// TIA Portal V17 export
// export: Created 2024-08-26T21:10:51.5472391Z, ExportSetting WithDefaults, DisplayName Totally Integrated Automation Portal, DisplayVersion V17 Update 7, DisplayName TIA Portal Openness, DisplayVersion V17 Update 7, DisplayName TIA Portal Version Control Interface, DisplayVersion V17, DisplayName SINAMICS Startdrive Advanced, DisplayVersion V17 SP2, DisplayName SINAMICS Startdrive G110M, G120, G120C, G120D, G120P, G115D, DisplayVersion V17 SP2, DisplayName SINAMICS Startdrive G130, G150, S120, S150, SINAMICS MV, S210, DisplayVersion V17 SP2, DisplayName STEP 7 Professional, DisplayVersion V17 Update 7, DisplayName STEP 7 Safety, DisplayVersion V17 Update 6, DisplayName WinCC Advanced / Unified PC, DisplayVersion V17 Update 7
FUNCTION "MODE" : Void   // FC4, LAD
{ S7_Optimized_Access := 'TRUE' }
VERSION : 0.1
// stored: AutoNumber true, IsIECCheckEnabled false, SetENOAutomatically false, UDAEnableTagReadback false
   VAR_TEMP
      f7 : Bool;
      BF7 : Bool;
   END_VAR
BEGIN

REGION Network 1: MODE CHANGE
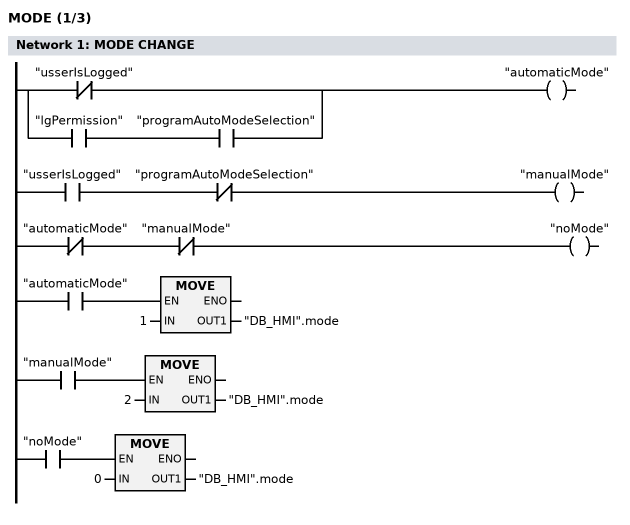
   RUNG wire#powerrail
      I_Contact( "usserIsLogged" )
      wire#w1
      Coil( "automaticMode" )
   END_RUNG
   RUNG wire#powerrail
      Contact( "lgPermission" )
      Contact( "programAutoModeSelection" )
   END_RUNG wire#w1
   RUNG wire#powerrail
      Contact( "usserIsLogged" )
      I_Contact( "programAutoModeSelection" )
      Coil( "manualMode" )
   END_RUNG
   RUNG wire#powerrail
      I_Contact( "automaticMode" )
      I_Contact( "manualMode" )
      Coil( "noMode" )
   END_RUNG
   RUNG wire#powerrail
      Contact( "automaticMode" )
      Move(in := 1, out1 => "DB_HMI".mode)
   END_RUNG
   RUNG wire#powerrail
      Contact( "manualMode" )
      Move(in := 2, out1 => "DB_HMI".mode)
   END_RUNG
   RUNG wire#powerrail
      Contact( "noMode" )
      Move(in := 0, out1 => "DB_HMI".mode)
   END_RUNG
   // the same network as SCL:
   "automaticMode" := NOT "usserIsLogged" OR ("lgPermission" AND "programAutoModeSelection");
   "manualMode" := "usserIsLogged" AND NOT "programAutoModeSelection";
   "noMode" := NOT "automaticMode" AND NOT "manualMode";
   IF "automaticMode" THEN "DB_HMI".mode := 1; END_IF;
   IF "manualMode" THEN "DB_HMI".mode := 2; END_IF;
   IF "noMode" THEN "DB_HMI".mode := 0; END_IF;
END_REGION

REGION Network 2: MODEL SELECTION
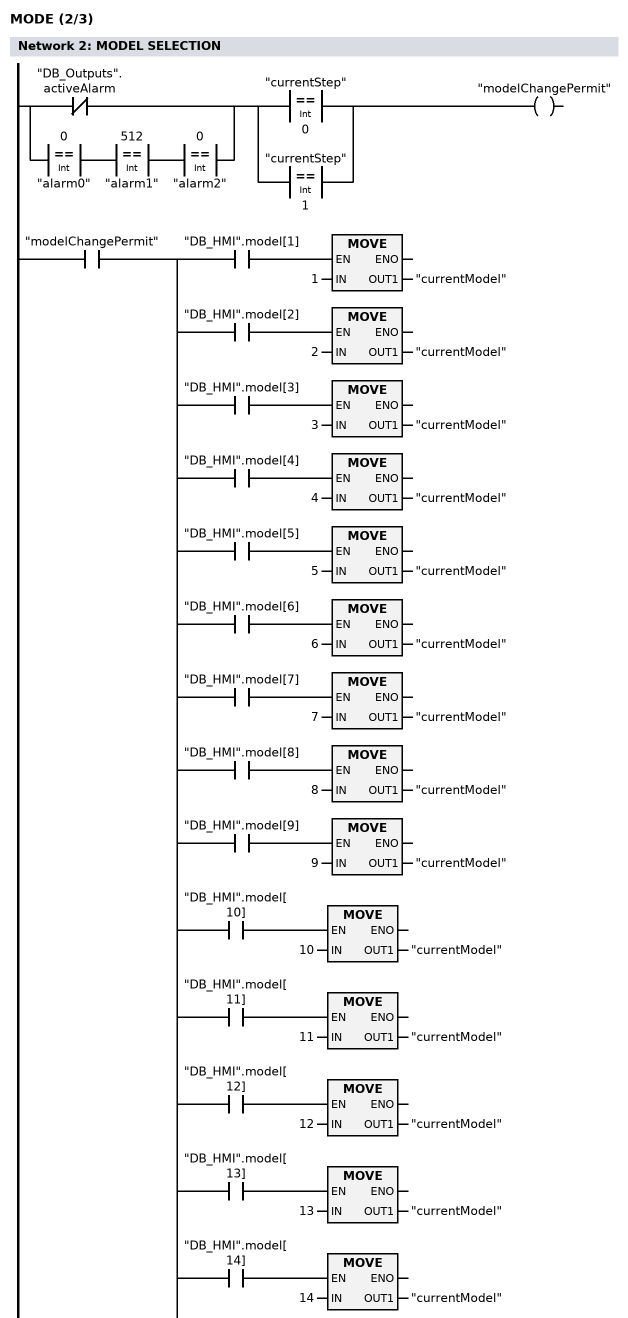
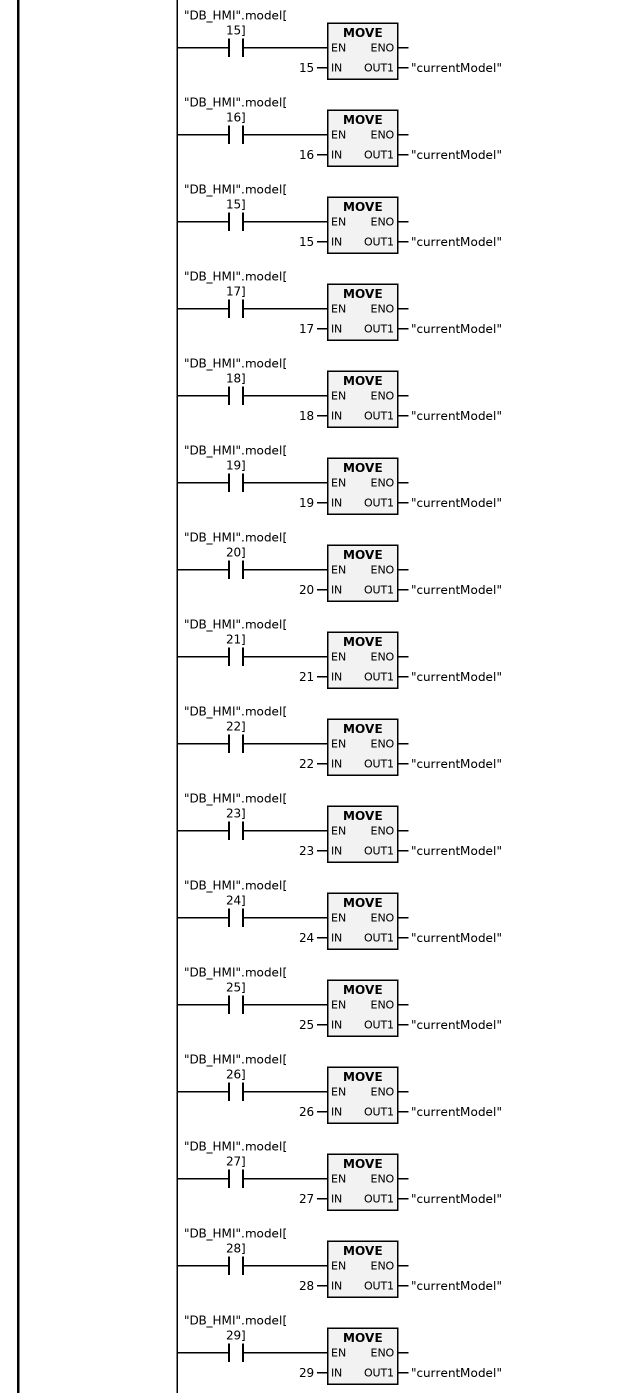
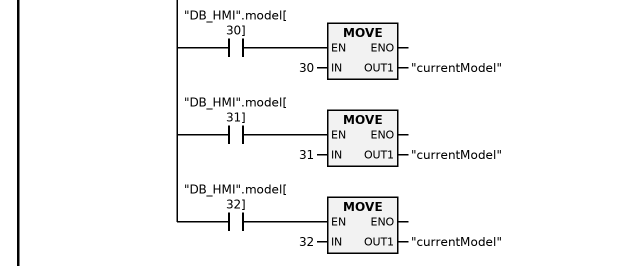
   RUNG wire#powerrail
      I_Contact( "DB_Outputs".activeAlarm )
      wire#w1
      { S7_Templates := "SrcType := Int" } EQ_Contact(in1 := "currentStep", in2 := 0)
      wire#w2
      Coil( "modelChangePermit" )
   END_RUNG
   RUNG wire#powerrail
      { S7_Templates := "SrcType := Int" } EQ_Contact(in1 := 0, in2 := "alarm0")
      { S7_Templates := "SrcType := Int" } EQ_Contact(in1 := 512, in2 := "alarm1")
      { S7_Templates := "SrcType := Int" } EQ_Contact(in1 := 0, in2 := "alarm2")
   END_RUNG wire#w1
   RUNG wire#w1
      { S7_Templates := "SrcType := Int" } EQ_Contact(in1 := "currentStep", in2 := 1)
   END_RUNG wire#w2
   RUNG wire#powerrail
      Contact( "modelChangePermit" )
      wire#w3
      Contact( "DB_HMI".model[1] )
      Move(in := 1, out1 => "currentModel")
   END_RUNG
   RUNG wire#w3
      Contact( "DB_HMI".model[2] )
      Move(in := 2, out1 => "currentModel")
   END_RUNG
   RUNG wire#w3
      Contact( "DB_HMI".model[3] )
      Move(in := 3, out1 => "currentModel")
   END_RUNG
   RUNG wire#w3
      Contact( "DB_HMI".model[4] )
      Move(in := 4, out1 => "currentModel")
   END_RUNG
   RUNG wire#w3
      Contact( "DB_HMI".model[5] )
      Move(in := 5, out1 => "currentModel")
   END_RUNG
   RUNG wire#w3
      Contact( "DB_HMI".model[6] )
      Move(in := 6, out1 => "currentModel")
   END_RUNG
   RUNG wire#w3
      Contact( "DB_HMI".model[7] )
      Move(in := 7, out1 => "currentModel")
   END_RUNG
   RUNG wire#w3
      Contact( "DB_HMI".model[8] )
      Move(in := 8, out1 => "currentModel")
   END_RUNG
   RUNG wire#w3
      Contact( "DB_HMI".model[9] )
      Move(in := 9, out1 => "currentModel")
   END_RUNG
   RUNG wire#w3
      Contact( "DB_HMI".model[10] )
      Move(in := 10, out1 => "currentModel")
   END_RUNG
   RUNG wire#w3
      Contact( "DB_HMI".model[11] )
      Move(in := 11, out1 => "currentModel")
   END_RUNG
   RUNG wire#w3
      Contact( "DB_HMI".model[12] )
      Move(in := 12, out1 => "currentModel")
   END_RUNG
   RUNG wire#w3
      Contact( "DB_HMI".model[13] )
      Move(in := 13, out1 => "currentModel")
   END_RUNG
   RUNG wire#w3
      Contact( "DB_HMI".model[14] )
      Move(in := 14, out1 => "currentModel")
   END_RUNG
   RUNG wire#w3
      Contact( "DB_HMI".model[15] )
      Move(in := 15, out1 => "currentModel")
   END_RUNG
   RUNG wire#w3
      Contact( "DB_HMI".model[16] )
      Move(in := 16, out1 => "currentModel")
   END_RUNG
   RUNG wire#w3
      Contact( "DB_HMI".model[15] )
      Move(in := 15, out1 => "currentModel")
   END_RUNG
   RUNG wire#w3
      Contact( "DB_HMI".model[17] )
      Move(in := 17, out1 => "currentModel")
   END_RUNG
   RUNG wire#w3
      Contact( "DB_HMI".model[18] )
      Move(in := 18, out1 => "currentModel")
   END_RUNG
   RUNG wire#w3
      Contact( "DB_HMI".model[19] )
      Move(in := 19, out1 => "currentModel")
   END_RUNG
   RUNG wire#w3
      Contact( "DB_HMI".model[20] )
      Move(in := 20, out1 => "currentModel")
   END_RUNG
   RUNG wire#w3
      Contact( "DB_HMI".model[21] )
      Move(in := 21, out1 => "currentModel")
   END_RUNG
   RUNG wire#w3
      Contact( "DB_HMI".model[22] )
      Move(in := 22, out1 => "currentModel")
   END_RUNG
   RUNG wire#w3
      Contact( "DB_HMI".model[23] )
      Move(in := 23, out1 => "currentModel")
   END_RUNG
   RUNG wire#w3
      Contact( "DB_HMI".model[24] )
      Move(in := 24, out1 => "currentModel")
   END_RUNG
   RUNG wire#w3
      Contact( "DB_HMI".model[25] )
      Move(in := 25, out1 => "currentModel")
   END_RUNG
   RUNG wire#w3
      Contact( "DB_HMI".model[26] )
      Move(in := 26, out1 => "currentModel")
   END_RUNG
   RUNG wire#w3
      Contact( "DB_HMI".model[27] )
      Move(in := 27, out1 => "currentModel")
   END_RUNG
   RUNG wire#w3
      Contact( "DB_HMI".model[28] )
      Move(in := 28, out1 => "currentModel")
   END_RUNG
   RUNG wire#w3
      Contact( "DB_HMI".model[29] )
      Move(in := 29, out1 => "currentModel")
   END_RUNG
   RUNG wire#w3
      Contact( "DB_HMI".model[30] )
      Move(in := 30, out1 => "currentModel")
   END_RUNG
   RUNG wire#w3
      Contact( "DB_HMI".model[31] )
      Move(in := 31, out1 => "currentModel")
   END_RUNG
   RUNG wire#w3
      Contact( "DB_HMI".model[32] )
      Move(in := 32, out1 => "currentModel")
   END_RUNG
   // the same network as SCL:
   "modelChangePermit" := (NOT "DB_Outputs".activeAlarm OR ((0 = "alarm0") AND (512 = "alarm1") AND (0 = "alarm2"))) AND (("currentStep" = 0) OR ("currentStep" = 1));
   IF "modelChangePermit" AND "DB_HMI".model[1] THEN "currentModel" := 1; END_IF;
   IF "modelChangePermit" AND "DB_HMI".model[2] THEN "currentModel" := 2; END_IF;
   IF "modelChangePermit" AND "DB_HMI".model[3] THEN "currentModel" := 3; END_IF;
   IF "modelChangePermit" AND "DB_HMI".model[4] THEN "currentModel" := 4; END_IF;
   IF "modelChangePermit" AND "DB_HMI".model[5] THEN "currentModel" := 5; END_IF;
   IF "modelChangePermit" AND "DB_HMI".model[6] THEN "currentModel" := 6; END_IF;
   IF "modelChangePermit" AND "DB_HMI".model[7] THEN "currentModel" := 7; END_IF;
   IF "modelChangePermit" AND "DB_HMI".model[8] THEN "currentModel" := 8; END_IF;
   IF "modelChangePermit" AND "DB_HMI".model[9] THEN "currentModel" := 9; END_IF;
   IF "modelChangePermit" AND "DB_HMI".model[10] THEN "currentModel" := 10; END_IF;
   IF "modelChangePermit" AND "DB_HMI".model[11] THEN "currentModel" := 11; END_IF;
   IF "modelChangePermit" AND "DB_HMI".model[12] THEN "currentModel" := 12; END_IF;
   IF "modelChangePermit" AND "DB_HMI".model[13] THEN "currentModel" := 13; END_IF;
   IF "modelChangePermit" AND "DB_HMI".model[14] THEN "currentModel" := 14; END_IF;
   IF "modelChangePermit" AND "DB_HMI".model[15] THEN "currentModel" := 15; END_IF;
   IF "modelChangePermit" AND "DB_HMI".model[16] THEN "currentModel" := 16; END_IF;
   IF "modelChangePermit" AND "DB_HMI".model[15] THEN "currentModel" := 15; END_IF;
   IF "modelChangePermit" AND "DB_HMI".model[17] THEN "currentModel" := 17; END_IF;
   IF "modelChangePermit" AND "DB_HMI".model[18] THEN "currentModel" := 18; END_IF;
   IF "modelChangePermit" AND "DB_HMI".model[19] THEN "currentModel" := 19; END_IF;
   IF "modelChangePermit" AND "DB_HMI".model[20] THEN "currentModel" := 20; END_IF;
   IF "modelChangePermit" AND "DB_HMI".model[21] THEN "currentModel" := 21; END_IF;
   IF "modelChangePermit" AND "DB_HMI".model[22] THEN "currentModel" := 22; END_IF;
   IF "modelChangePermit" AND "DB_HMI".model[23] THEN "currentModel" := 23; END_IF;
   IF "modelChangePermit" AND "DB_HMI".model[24] THEN "currentModel" := 24; END_IF;
   IF "modelChangePermit" AND "DB_HMI".model[25] THEN "currentModel" := 25; END_IF;
   IF "modelChangePermit" AND "DB_HMI".model[26] THEN "currentModel" := 26; END_IF;
   IF "modelChangePermit" AND "DB_HMI".model[27] THEN "currentModel" := 27; END_IF;
   IF "modelChangePermit" AND "DB_HMI".model[28] THEN "currentModel" := 28; END_IF;
   IF "modelChangePermit" AND "DB_HMI".model[29] THEN "currentModel" := 29; END_IF;
   IF "modelChangePermit" AND "DB_HMI".model[30] THEN "currentModel" := 30; END_IF;
   IF "modelChangePermit" AND "DB_HMI".model[31] THEN "currentModel" := 31; END_IF;
   IF "modelChangePermit" AND "DB_HMI".model[32] THEN "currentModel" := 32; END_IF;
END_REGION

REGION Network 3: GAP LEADER HMI MODE
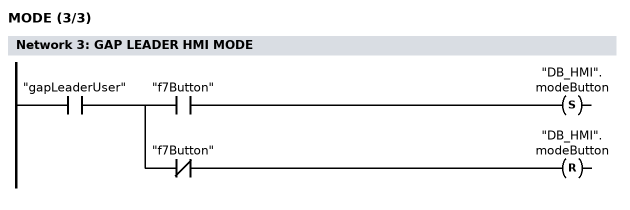
   RUNG wire#powerrail
      Contact( "gapLeaderUser" )
      wire#w1
      Contact( "f7Button" )
      S_Coil( "DB_HMI".modeButton )
   END_RUNG
   RUNG wire#w1
      I_Contact( "f7Button" )
      R_Coil( "DB_HMI".modeButton )
   END_RUNG
   // the same network as SCL:
   IF "gapLeaderUser" AND "f7Button" THEN "DB_HMI".modeButton := TRUE; END_IF;
   IF "gapLeaderUser" AND NOT "f7Button" THEN "DB_HMI".modeButton := FALSE; END_IF;
END_REGION
END_FUNCTION
